// TIA Portal V20 export
// export: Created 2026-07-14T14:38:58.6437464Z, ExportSetting WithDefaults, DisplayName Totally Integrated Automation Portal, DisplayVersion V20 Update 5, DisplayName TIA Portal Openness, DisplayVersion V20 Update 4, DisplayName TIA Portal Version Control Interface, DisplayVersion V20 Update 5, DisplayName SINAMICS Startdrive Advanced, DisplayVersion V20, DisplayName SINAMICS DCC, DisplayVersion V20, DisplayName SINAMICS Startdrive G130, G150, S120, S150, SINAMICS MV, G220, S200, S210, DisplayVersion V20, DisplayName SINAMICS Startdrive G110M, G120, G120C, G120D, G120P, G115D, DisplayVersion V20, DisplayName STEP 7 Professional, DisplayVersion V20 Update 5, DisplayName STEP 7 Safety, DisplayVersion V20 Update 2, DisplayName WinCC Basic/Comfort/Advanced, DisplayVersion V20 Update 5, DisplayName WinCC Unified, DisplayVersion V20 Update 5
FUNCTION "ScaleValue" : Void   // FC25, LAD
{ S7_Optimized_Access := 'TRUE' }
VERSION : 0.1
// Reference callee FC for CALL examples (TimingAndCalls)
// stored: AutoNumber true, IsIECCheckEnabled false, SetENOAutomatically false, UDAEnableTagReadback false
   VAR_INPUT
      RawInput : Real;
      ScaleFactor : Real;
   END_VAR
   VAR_OUTPUT
      ScaledResult : Real;
   END_VAR
BEGIN

REGION Network 1: Linear scale
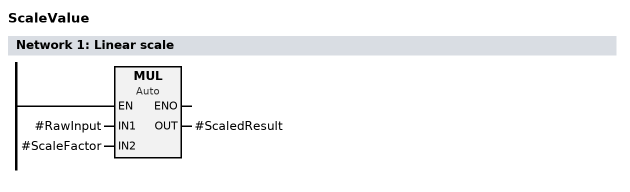
   RUNG wire#powerrail
      Mul(in1 := #RawInput, in2 := #ScaleFactor, out => #ScaledResult)
   END_RUNG
   // the same network as SCL:
   #ScaledResult := #RawInput * #ScaleFactor;
END_REGION
END_FUNCTION
